TYPE EL2014_Outputs :
STRUCT
	{attribute addProperty Name "Channel 1"}
	_1 AT %Q* : DIGOutput;
	{attribute addProperty Name "Channel 2"}
	_2 AT %Q* : DIGOutput;
	{attribute addProperty Name "Channel 3"}
	_3 AT %Q* : DIGOutput;
	{attribute addProperty Name "Channel 4"}
	_4 AT %Q* : DIGOutput;
END_STRUCT
END_TYPE

(* stored: Version 1.1.0.1, ProductVersion 3.1.4024.9
   DUT EL2014_Outputs: Id {6e6b36d4-7a6f-014a-3e11-e7cc8ace6ba4} *)
